(* CoDeSys 2.3 export: TXQUEUE_10.EXP *)

(* Data type *)
TYPE TxQueue_10 :
STRUCT
	TxCounter      : UINT;
	RxCounter      : UINT;
	NoOfTxMessages : UINT;
	TxMessages     : ARRAY [0..9] OF ARRAY[0..13] OF BYTE;
END_STRUCT
END_TYPE
